FUNCTION_BLOCK FB_RunCyclicTasksAction EXTENDS FB_Action
VAR
END_VAR

METHOD  Execute
VAR_INPUT
    ipObject: I_Object;
END_VAR
VAR
    ipTask: I_CyclicTask;
END_VAR
IF __QUERYINTERFACE(ipObject, ipTask) THEN
    ipTask.Run();
END_IF
END_METHOD

END_FUNCTION_BLOCK

(* stored: Version 1.1.0.1, ProductVersion 3.1.4024.12
   POU FB_RunCyclicTasksAction: Id {36e0149e-be33-0243-3d91-faad07c1f86d}, SpecialFunc None
   Method Execute: Id {9ab3fc93-83ee-0789-0ca2-c5a70700af2e} *)
